(* IEC 61131-3 sources: BLM_BACKGROUND/src/PROGRAM_FILES/FB (part 5) *)

              //Modifica per gestione override come limitazione e non come percentuale
              ovr:=(i_sys_hwOvr_appo*i_sys_swOvr)/100;
              IF ovr>i_sys_tOVR THEN
                  ovr:=i_sys_tOVR;
              END_IF;
            //   {#ifdef PROFINET}
            //       {#ifndef ORBITALE}
                      IF TestVelHoldToRun()=TRUE AND i_sys_OPMODE=AUTOMODE AND FlgRiduzVelVGP=FALSE AND (TestMasterLavoro()=TRUE OR FlgPezzoInEsecuzione=TRUE) THEN
                          //Impostazione override per gestione hold TO run in automatico immediatamente al termine del primo start, così
                          //che al momento di iniziare la movimentazione degli assi l^override attivo sia già impostato al valore definito
                          //nel parametro Q4100
                          IF ovr>i_sys_override_HoldToRun_Auto THEN
                              ovr:=i_sys_override_HoldToRun_Auto;
                          END_IF;
                      END_IF;
            //       {#endif}  //Fine NO ORBITALE
            //   {#endif}	//Fine PROFINET
              IF i_sys_stopcond<>0 THEN
                //   {#ifdef PROFINET}
                      IF (i_Barriera=FALSE OR i_sys_BarrieraViolata=TRUE) AND TEMPO_ARRESTO_BARRIERA>0.01 THEN
                          //In caso di violazione della barriera di sicurezza se definita
                          //si attiva l^apposita rampa di decelerazione
                          Appo:=TEMPO_ARRESTO_BARRIERA;
                          AccelerazioneMaster:=1/Appo;
                      ELSE
                          AccelerazioneMaster:=i_sys_acc_master;
                      END_IF;
                //   {#else}  //Fine PROFINET
                      IF i_sys_BarrieraViolata=TRUE AND TEMPO_ARRESTO_BARRIERA>0.01 THEN
                          //In caso di violazione della barriera di sicurezza se definita
                          //si attiva l^apposita rampa di decelerazione
                          Appo:=TEMPO_ARRESTO_BARRIERA;
                          AccelerazioneMaster:=1/Appo;
                      ELSE
                          AccelerazioneMaster:=i_sys_acc_master;
                      END_IF;
                //   {#endif}  //Fine NO PROFINET
                  i_sys_ovr:=0;
                  CURRENT_STATE:=_FB_MCP483#STATE_MCP483_STOP_ASSI_MASTER;
              ELSE
                //   {#ifdef ORBITALE}
                //       {#ifdef DH4010}
                          i_sys_ovr:=ovr;
                    //   {#else}  //Fine DH4010
                          IF i_sys_OPMODE=AUTOMODE THEN
                              IF TestMasterLavoro()=TRUE THEN
                                  IF getBit(TO_DWORD(ReadTabStati(Riga:=rc, Colonna:=COL_RESERVED1, Programma:=I_SYS_Current_Prog, Tabella:=SINT#-1)), TO_USINT(BIT_NO_OVERRIDE))=TRUE THEN
                                      //Gestione forzatura OVERRIDE nel ciclo automatico nelle linee della tabella
                                      //stati dove e^ previsto (ad esempio per il taglio)
                                      i_sys_ovr_act:=100;
                                      i_sys_ovr:=100;
                                      masteraxis:=AsPositioningAxisRef(Axes[X1].masteraxis);
                                      masteraxis^._override.velocity:=100;
                                  ELSE
                                      i_sys_ovr:=ovr;
                                  END_IF;
                              ELSE
                                  //Primo start
                                //   {#ifdef FOUR_RUNNER_PLAUNO}
                                      IF i_sys_OverrideMarcatura=TRUE THEN
                                          //Forzatura override al 100% per mantenere costante la lunghezza della scritta
                                          i_sys_ovr_act:=100;
                                          i_sys_ovr:=100;
                                          masteraxis:=AsPositioningAxisRef(Axes[X1].masteraxis);
                                          masteraxis^._override.velocity:=100;
                                          //Axes[X1].masteraxis._override.velocity:=100;
                                      ELSE
                                          //Ripristiono override al termine della marcatura
                                          i_sys_ovr:=ovr;
                                      END_IF;
                                //   {#else}	//Fine FOUR_RUNNER_PLAUNO
                                      i_sys_ovr:=ovr;
                                //   {#endif};    //Fine NO FOUR_RUNNER_PLAUNO
                              END_IF;
                          ELSE
                              i_sys_ovr:=ovr;
                          END_IF;
                //       {#endif}  //Fine NO DH4010
                //   {#else}  //Fine ORBITALE
                      i_sys_ovr:=ovr;
                //   {#endif}  //Fine NO ORBITALE
                  CURRENT_STATE:=_FB_MCP483#STATE_MCP483_READ_OVR_2;
              END_IF;

            _FB_MCP483#STATE_MCP483_STOP_ASSI_MASTER:
              IF StopAssiMaster.outputState<>GENERAL_STATE#STATE_END THEN
                  StopAssiMaster(AccelerazioneMaster:=AccelerazioneMaster (* , ProssimoComando:=IMMEDIATELY*));
              ELSE
                  StopAssiMaster();
                  CURRENT_STATE:=_FB_MCP483#STATE_MCP483_READ_OVR_2;
              END_IF;

            _FB_MCP483#STATE_MCP483_READ_OVR_2:
               {::ifndef MCP_1900}
                  //Legge il II Override
                  i_sys_hwOVR2:=read_ovr2(mcpi_spindleoverride_a,mcpi_spindleoverride_b,mcpi_spindleoverride_c,mcpi_spindleoverride_d);
                  ovr2:=((i_sys_hwOvr2)/100) * ((i_sys_swOvr2)/100) * 100;
                  IF i_sys_stopcond<>0 THEN
                      i_sys_ovr2:=0;
                  ELSE
                      i_sys_ovr2:=ovr2;
                  END_IF;
               {::else}	//FINE NO MCP_1900
                  IF i_sys_stopcond<>0 THEN
                      i_sys_ovr2:=0;
                  ELSE
                      i_sys_ovr2:=100;
                  END_IF;
            {::endif} //FINE MCP_1900
              ovr2:=((i_sys_hwOvr2)/100) * ((i_sys_swOvr2)/100) * 100;
              IF i_sys_stopcond<>0 THEN
                  i_sys_ovr2:=0;
              ELSE
                  i_sys_ovr2:=ovr2;
              END_IF;
              //Assegnazione override all^asse master, per fare in modo di gestire la velocità
              //degli assi collegati in camma
              IF i_sys_stopcond=0 THEN
                  //Non deve essere attivo lo stop ciclo, in quanto in quella fase
                  //l^arresto dell master avviene con un normale comando di stop, associato
                  //alla rampa di decelerazione definita nella variabile AccelerazioneMaster
                  IF ABS(GetMasterOverride()-i_sys_ovr)>0.9 AND TestMasterVeloc()=TRUE THEN
                      //Al cambio di override corrisponde una immediata impostazione dell^accelerazione
                      //dell^asse master pari a 3 (quindi siamo a 0.3 secondi di rampa)
                      //Questo per evitare che ad ogni gradino venga causata sugli assi veri una
                      //accelerazione/decelerazione troppo elevata
                      IF ABS(GetMasterMaxAcceleration()-ACCELERATION_MASTER)>0.1 THEN
                          SetMasterMaxAcceleration(Value:=ACCELERATION_MASTER);
                      END_IF;
                  ELSE
                      //Senza nessun cambio di override si ripristina l^accelerazione standard del master
                      //molto elavata
                      IF ABS(GetMasterMaxAcceleration()-MAX_MASTER_ACCELERATION)>0.1 THEN
                          SetMasterMaxAcceleration(Value:=MAX_MASTER_ACCELERATION);
                      END_IF;
                  END_IF;
                  //Impostazione dell^override dell^asse master
                  IF ABS(GetMasterOverride()-i_sys_ovr_Act)>0.001 THEN
                      SetMasterVelocity(Value:=i_sys_ovr_Act);
                    //   {#ifdef RUNNER}
                    //       {#ifdef FOUR_RUNNER_PLAUNO}
                    //           {#ifndef PLAUNO_LIGHT}
                                masteraxis:=AsPositioningAxisRef(Axes[A1].masteraxis);
                                masteraxis^._override.velocity:=i_sys_ovr_Act;
                        //       {#endif} //FINE NO PLAUNO_LIGHT
                        //   {#endif}  //Fine FOUR_RUNNER_PLAUNO
                        //   {#ifdef B1_B2}
                              masteraxis:=AsPositioningAxisRef(Axes[B1].masteraxis);
                              masteraxis^._override.velocity:=i_sys_ovr_Act;
                    //       {#endif}  //Fine B1_B2
                    //   {#endif}  //Fine RUNNER
                  END_IF;
              ELSE
                  //Lo stop ciclo è attivo
                  IF TestMasterVeloc()=FALSE THEN
                      //Con stop ciclo attivo si imposta l^override desiderato quando il master si è fermato
                      IF ABS(GetMasterOverride()-i_sys_ovr_Act)>0.001 THEN
                          SetMasterVelocity(Value:=i_sys_ovr_Act);
                        //   {#ifdef RUNNER}
                        //       {#ifdef FOUR_RUNNER_PLAUNO}
                        //           {#ifndef PLAUNO_LIGHT}
                                      masteraxis:=AsPositioningAxisRef(Axes[A1].masteraxis);
                                      masteraxis^._override.velocity:=i_sys_ovr_Act;
                            //       {#endif} //FINE NO PLAUNO_LIGHT
                            //   {#endif}  //Fine FOUR_RUNNER_PLAUNO
                            //   {#ifdef B1_B2}
                                    masteraxis:=AsPositioningAxisRef(Axes[B1].masteraxis);
                                    masteraxis^._override.velocity:=i_sys_ovr_Act;
                        //       {#endif}  //Fine B1_B2
                        //   {#endif}  //Fine RUNNER
                      END_IF;
                  END_IF;
                  //Lo stop ciclo si esegue con l^accelerazione standard del master
                  IF ABS(GetMasterMaxAcceleration()-MAX_MASTER_ACCELERATION)>0.1 THEN
                      SetMasterMaxAcceleration(Value:=MAX_MASTER_ACCELERATION);
                  END_IF;
              END_IF;
              FOR i:=_FIRST_AXIS#FIRST_AXIS TO _FIRST_AXIS#FIRST_AXIS+_MAXIS#MAXAXIS-1 BY 1 DO
                  IF CheckIfTOactive(Axis:=i)=TRUE THEN
                      //Se l^asse non è in CAMMA
                      PosAx:=AsSynchronousAxisRef(Axes[i].PosAx);
                      Camma:= AsCamRef(PosAx^.StatusSynchronizedMotion.ActualCam);
                      IF   PosAx^.StatusSynchronizedMotion.FunctionState <>3 THEN
                          {::ifdef AL_BLM}
                              IF i=L1 THEN
                                  //Essendo L1 un asse del caricatore, non deve essere gestito normalmente
                                  //in quanto deve consentire il funzionamento del caricatore, anche quando
                                  //l^override è impostato a 0 in quanto il dispositivo è fuori posizione
                                  IF i_sys_stopcond=1 THEN
                                    ;
                                      PosAx^._override.velocity:=i_sys_ovr_act;
                                  ELSE
                                    ;
                                      PosAx^._override.velocity:=i_sys_hwovr;
                                  END_IF;
                              ELSE
                            //     //   {#ifdef ASSE_Z2}
                                      IF i=Z2 THEN
                                        PosAx:=AsSynchronousAxisRef(Axes[i].PosAx);
                                          IF i_sys_stopcond=1 THEN ;
                                            PosAx^._override.velocity:=i_sys_ovr_act;
                                          ELSE ;
                                            PosAx^._override.velocity:=100;
                                          END_IF;
                                      ELSE ;
                                            PosAx^._override.velocity:=i_sys_ovr_act;
                                      END_IF;
                                //   {#else}  //Fine ASSE_Z2
                                            PosAx^._override.velocity:=i_sys_ovr_act;
                                //   {#endif}  //Fine NO ASSE_Z2
                              END_IF;
                          {::else}  //Fine AL_BLM
                        //       {#ifdef EFLEX}
                                  IF i=W1 THEN
                                        PosAx:=AsSynchronousAxisRef(Axes[i].PosAx);
                                      IF (i_sys_OpMode=JOGMODE AND i_sys_activedevice=CMD_TAGLIO_EFLEX) OR
                                           (i_sys_OpMode=AUTOMODE AND PosizioneMaster()=POSIZIONE_MASTER_RFI) THEN
                                          //Asse W1 (trancia) non deve sentire override quando taglia con
                                          //il comando manuale
                                          PosAx^._override.velocity:=100;
                                      ELSE
                                          PosAx^._override.velocity:=i_sys_ovr_act;
                                      END_IF;
                                  ELSE
                                      //Gestione standard asse
                                      PosAx^._override.velocity:=i_sys_ovr_act;
                                  END_IF;
                            //   {#else}  //Fine EFLEX
                            //       {#ifdef RUNNER}
                            //           {#ifdef FOUR_RUNNER_PLAUNO}
                            //               {#ifdef B1_B2}
                                            //   IF {#ifndef PLAUNO_LIGHT}i=A1 OR i=A2 OR {#endif} i=B1 OR i=B2 THEN
                                            //       IF i_sys_ovr_act>0.1 THEN
                                            //           assi[i].PosAx._override.velocity:=100;
                                            //       ELSE
                                            //           assi[i].PosAx._override.velocity:=i_sys_ovr_act;
                                            //       END_IF;
                                            //   ELSE
                                            //       //Gestione standard asse
                                            //       assi[i].PosAx._override.velocity:=i_sys_ovr_act;
                                            //   END_IF;
                                        //   {#else}  //Fine B1_B2
                                        //       {#ifndef PLAUNO_LIGHT}
                                                  IF i=A1 OR i=A2 THEN
                                                    PosAx:=AsSynchronousAxisRef(Axes[i].PosAx);
                                                      IF i_sys_ovr_act>0.1 THEN ;
                                                          //PosAx^._override.velocity:=100;
                                                      ELSE ;
                                                          //PosAx^._override.velocity:=i_sys_ovr_act;
                                                      END_IF;
                                                  ELSE ;
                                            //   {#endif} //FINE NO PLAUNO_LIGHT
                                              //Gestione standard asse
                                                   // PosAx^._override.velocity:=i_sys_ovr_act;
                                            //   {#ifndef PLAUNO_LIGHT}
                                                  END_IF;
                                    //           {#endif}	//Fine PLAUNO_LIGHT
                                    //       {#endif}  //Fine NO B1_B2
                                    //   {#endif}  //Fine FOUR_RUNNER_PLAUNO
                                    //   {#ifdef THREE_RUNNER_TWO_RUNNER}
                                    //       {#ifdef B1_B2}
                                              IF i=A1 OR i=B1 OR i=B2 THEN
                                                PosAx:=AsSynchronousAxisRef(Axes[i].PosAx);
                                                  IF i_sys_ovr_act>0.1 THEN ;
                                                      //PosAx^._override.velocity:=100;
                                                  ELSE ;
                                                      //PosAx^._override.velocity:=i_sys_ovr_act;
                                                  END_IF;
                                              ELSE ;
                                                  //Gestione standard asse
                                                  //PosAx^._override.velocity:=i_sys_ovr_act;
                                              END_IF;
                                        //   {#else}  //Fine B1_B2
                                              IF i=A1 THEN
                                                  IF i_sys_ovr_act>0.1 THEN ;
                                                      //PosAx^._override.velocity:=100;
                                                  ELSE ;
                                                      //PosAx^._override.velocity:=i_sys_ovr_act;
                                                  END_IF;
                                              ELSE ;
                                                  //Gestione standard asse
                                                  //PosAx^._override.velocity:=i_sys_ovr_act;
                                              END_IF;
                                //           {#endif}  //Fine NO B1_B2
                                //       {#endif}  //Fine THREE_RUNNER_TWO_RUNNER
                                //   {#else}  //Fine RUNNER
                                      //Gestione standard asse
                                      //PosAx^._override.velocity:=i_sys_ovr_act;
                        //           {#endif}  //Fine NO RUNNER
                        //       {#endif}  //Fine NO EFLEX
                          {::endif}  //Fine NO AL_BLM
                          ;
                      END_IF;
                  END_IF;
              END_FOR;
              //Assegna l^override agli oggetti interpolatore
              {::ifndef ORBITALE}
                KinAxesX1_U2_def:= KinAxesX1_U2;
                X1_U2:= AsKinematicsRef(KinAxesX1_U2_def);
                X1_U2^._override.velocity:=i_sys_ovr_act;
              {::endif}  //Fine ORBITALE
                //{::ifndef ETURN}
                    // {::ifndef ORBITALE}
                    //   {::ifndef ELECTMRL}
                    //         KinAxesW3_W4_Q1_def:= KinAxesW3_W4_Q1;
                    //         W3_W4_Q1:= AsKinematicsRef(KinAxesW3_W4_Q1_def);
                    //       W3_W4_Q1^._override.velocity:=i_sys_ovr_act;
                    // //   {#else}
                    //         KinAxesW3_W4_W6_Q1_def:= KinAxesW3_W4_W6_Q1;
                    //         W3_W4_W6_Q1:= AsKinematicsRef(KinAxesW3_W4_W6_Q1_def);
                    //         W3_W4_W6_Q1^._override.velocity:=i_sys_ovr_act;
            //           {#endif} //FINE ELECTMRL
            //       {#endif}	//Fine ORBITALE
            //   {#endif}  //Fine ETURN
            //   {#ifdef INTERPOLA_Y1_X1}
                  //Y1_X1._override.velocity:=i_sys_ovr_act;//
            //   {#endif}    //Fine INTERPOLA_Y1_X1
            //   {#ifdef INTERPOLA_X1_Y1}
                  //X1_Y1._override.velocity:=i_sys_ovr_act;//
            //   {#endif}	//Fine INTERPOLA_X1_Y1
            //   {#ifdef INTERPOLA_X2_Y2}
                  //X2_Y2._override.velocity:=i_sys_ovr_act;//
            //   {#endif}	//Fine INTERPOLA_X2_Y2
            //   {#ifdef INTERPOLA_X3_X6}
                  //X3_X6._override.velocity:=i_sys_ovr_act;//
            //   {#endif}	//Fine INTERPOLA_X3_X6
            //   {#ifdef INTERPOLA_X2_X6}
                  //X2_X6._override.velocity:=i_sys_ovr_act;//
            //   {#endif}	//Fine INTERPOLA_X2_X6
            {::ifdef SLITTA_MOBILE_DX}
             KinAxesY1_U4_def:= KinAxesY1_U4;
             Y1_U4:= AsKinematicsRef(KinAxesY1_U4_def);
             Y1_U4^._override.velocity:=i_sys_ovr_act;
                  //Y1_U4._override.velocity:=i_sys_ovr_act;//
            {::endif}	//Fine SLITTA_MOBILE_DX
            //   {#ifdef SLITTA_MOBILE_SX}
                  //Y1_U5._override.velocity:=i_sys_ovr_act;//
            //   {#endif}	//Fine SLITTA_MOBILE_SX
            //    {::ifdef MATRICE_ELETTRICA}
            //       IF TestAxesY2()=TRUE THEN
            //           Y1_U4_Y2._override.velocity:=i_sys_ovr_act;//
            //            Y1_Y2._override.velocity:=i_sys_ovr_act;//
            //        END_IF;
            //    {::endif}  //Fine MATRICE_ELETTRICA
            //   {#ifdef SOLLEVAMENTO_SLITTA_SPALLAMENTO}
                //   Q1_V1_V4._override.velocity:=i_sys_ovr_act;//
                //   Q1_V1._override.velocity:=i_sys_ovr_act;
            //   {#endif}	//Fine SOLLEVAMENTO_SLITTA_SPALLAMENTO
               {::ifdef INTERPOLA_Q1_V1_Z1}
            KinAxesQ1_V1_Z1_def:= KinAxesQ1_V1_Z1;
            Q1_V1_Z1:= AsKinematicsRef(KinAxesY1_U4_def);
            Q1_V1_Z1^._override.velocity:=i_sys_ovr_act;
                  //Q1_V1_Z1._override.velocity:=i_sys_ovr_act;
               {::endif}    //Fine INTERPOLA_Q1_V1_Z1
              IF i_sys_current_prog>=0 THEN
                  //Rinfresca il MASTER
                  SetPosizioneMaster(Programma:=i_sys_current_prog);
              END_IF;
              CURRENT_AXIS:=_FIRST_AXIS#FIRST_AXIS-1;
              CURRENT_STATE:= _FB_MCP483#STATE_MCP483_LOOP_HOMING;

        _FB_MCP483#STATE_MCP483_LOOP_HOMING:
              FOR i:=CURRENT_AXIS+1 TO _MAXIS#MAXAXIS-1 BY 1 DO
                  IF TestToAttivo(Asse:=i)=TRUE THEN
                    PosAx:=AsSynchronousAxisRef(Axes[i].PosAx);
                      IF  Posax^.StatusWord.%x1 = TRUE THEN
                          IF Posax^.ErrorDetail.Reaction<>0 THEN
                              //Ferma tutti gli altri assi
                              i_sys_stopcond:=1;
                              IF Posax^.StatusWord.%X0=TRUE THEN
                                  Abort_All();
                              END_IF;
                          END_IF;
                      END_IF;

                      //Verifica eventuali errori di creazione della camma
                      IF PosAx^.StatusSynchronizedMotion.ActualMaster <> UDINT#0 THEN
                     // IF Axes[i].sincroasse.activemaster<> NULL THEN
                        Camma:= AsCamRef(Axes[i].Camma);
                            IF Camma^.StatusWord.%X1 =TRUE THEN
                            //IF Axes[i].Camma.error=YES THEN
                               IF Camma^.ErrorDetail.Reaction <> 0 THEN
                              //IF assi[i].Camma.errorreaction<>NONE THEN
                                  i_sys_stopcond:=1;
                                    IF Posax^.StatusWord.%X0=TRUE THEN
                                  //IF assi[i].Posax.control=ACTIVE THEN
                                      Abort_All();
                                  END_IF;
                              END_IF;
                          END_IF;
                      END_IF;
                      IF posax^.VirtualAxis.Mode = UDINT#0 THEN
                          IF pm[i].ma_verifica_num_serie_encoder=TRUE THEN
                              Axes[i].Homed:=Axes[i].numserieencoder=pm[i].ma_num_serie_encoder AND
                                                           Axes[i].numserieencoder>0 AND
                                                           PosAx^.StatusWord.%X5= TRUE AND
                                                           pm[i].ma_stato_index=2;
                          ELSE
                              Axes[i].Homed:=PosAx^.StatusWord.%X5=TRUE AND
                                                           pm[i].ma_stato_index=2;
                        ;  END_IF;
                      ELSE
                          IF PosAx^.StatusWord.%X5=TRUE THEN
                              //Asse virtuale l^asse viene indexato di default
                              pm[i].ma_stato_index:=SINT#0;
                              CURRENT_AXIS:=i;
                              CURRENT_STATE:=_FB_MCP483#STATE_MCP483_LOOP_HOMING_ABSOLUTE;
                              EXIT;
                          END_IF;
                      END_IF;
                  END_IF;
              END_FOR;
              IF CURRENT_STATE<>_FB_MCP483#STATE_MCP483_LOOP_HOMING_ABSOLUTE THEN
                  CURRENT_STATE:=_FB_MCP483#STATE_MCP483_CHECK_HOMING_ERRORS;
              END_IF;

            //   CURRENT_AXIS:=CURRENT_AXIS+1;
            //   IF CURRENT_AXIS<_MAXIS#MAXAXIS THEN
            //     PosAx:= AsSynchronousAxisRef(Axes[CURRENT_AXIS].Posax);
            //       IF TestToAttivo(Asse:=CURRENT_AXIS)=TRUE THEN
            //           IF Posax^.ErrorWord=TRUE THEN
            //             IF Posax^.ErrorDetail.Reaction<>0 THEN
            //               //IF assi[CURRENT_AXIS].Posax.errorreaction<>NONE THEN
            //                   //Ferma tutti gli altri assi
            //                   i_sys_stopcond:=1;
            //                   IF Posax^.StatusWord.%X0=TRUE THEN
            //                   //IF assi[CURRENT_AXIS].Posax.control=ACTIVE THEN
            //                       Abort_All();
            //                   END_IF;
            //               END_IF;
            //           END_IF;
            //           sincroasse:= AsSynchronousAxisRef( assi[CURRENT_AXIS].Sincroasse);
            //           IF Sincroasse^.ErrorWord=TRUE THEN
            //           //IF.error=YES THEN
            //             IF Sincroasse^.ErrorDetail.Reaction<>0 THEN
            //               //IF Sincroasse^.errorreaction<>NONE THEN
            //                   i_sys_stopcond:=1;
            //                   PosAx:= AsSynchronousAxisRef(Axes[i].Posax);
            //                   IF Posax^.StatusWord.%X0=TRUE THEN
            //                       Abort_All();
            //                   END_IF;
            //               END_IF;
            //           END_IF;
            //           //Verifica eventuali errori di creazione della camma
            //           sincroasse:= AsSynchronousAxisRef(Axes[CURRENT_AXIS].sincroasse);
            //           IF sincroasse^.StatusSynchronizedMotion.ActualMaster <> UDINT#0 THEN
            //           //IF Axes[CURRENT_AXIS].sincroasse.activemaster<>NULL THEN
            //           Camma:= AsCamRef(Axes[i].Camma);
            //           IF Camma^.ErrorWord=TRUE THEN
            //           //IF Axes[i].Camma.error=YES THEN
            //              IF Camma^.ErrorDetail.Reaction <> 0 THEN
            //               //IF assi[CURRENT_AXIS].Camma.error=YES THEN
            //                   //IF assi[CURRENT_AXIS].Camma.errorreaction<>NONE THEN
            //                       i_sys_stopcond:=1;
            //                       IF assi[CURRENT_AXIS].Posax.control=ACTIVE THEN
            //                           Abort_All();
            //                       END_IF;
            //                   END_IF;
            //               END_IF;
            //           END_IF;
            //           IF Axes[CURRENT_AXIS].posax.typeofaxis<>VIRTUAL_AXIS THEN
            //               IF pm[CURRENT_AXIS].ma_verifica_num_serie_encoder=TRUE THEN
            //                   Axes[CURRENT_AXIS].Homed:=Axes[CURRENT_AXIS].numserieencoder=pm[CURRENT_AXIS].ma_num_serie_encoder AND
            //                                                Axes[CURRENT_AXIS].numserieencoder>0 AND
            //                                                Axes[CURRENT_AXIS].PosAx.positioningstate.homed=YES AND
            //                                                pm[CURRENT_AXIS].ma_stato_index=2;
            //               ELSE
            //                   Axes[CURRENT_AXIS].Homed:=Axes[CURRENT_AXIS].PosAx.positioningstate.homed=YES AND
            //                                                pm[CURRENT_AXIS].ma_stato_index=2;
            //               END_IF;
            //           ELSE
            //               IF Axes[CURRENT_AXIS].PosAx.positioningstate.homed<>YES THEN
            //                   //Asse virtuale l^asse viene indexato di default
            //                   pm[CURRENT_AXIS].ma_stato_index:=0;
            //                   CURRENT_STATE:=STATE_MCP483_LOOP_HOMING_HOMING_ABSOLUTE;
            //               END_IF;
            //           END_IF;
            //       END_IF;
            //   ELSE
            //       CURRENT_STATE:=_FB_MCP483#STATE_MCP483_CHECK_HOMING_ERRORS;
            //   END_IF;

          _FB_MCP483#STATE_MCP483_LOOP_HOMING_ABSOLUTE:
              IF Homing_Absolute.outputState<>GENERAL_STATE#STATE_END THEN
                  Homing_absolute(Asse:=CURRENT_AXIS, Position:=0);
              ELSE
                  Homing_absolute();
                  Axes[CURRENT_AXIS].homed:=TRUE;
                  CURRENT_STATE:=_FB_MCP483#STATE_MCP483_LOOP_HOMING;
              END_IF;

          _FB_MCP483#STATE_MCP483_CHECK_HOMING_ERRORS:
            //   {#ifdef INTERPOLA_Y1_X1}
                //   IF Y1_X1.error=YES THEN %%%%
                //       IF Y1_X1.errorreaction<>NONE THEN
                //           //Ferma tutti gli altri assi
                //           i_sys_stopcond:=1;
                //           IF Y1_X1.linearPathCommand.state=ACTIVE THEN //OT.StatusWord.%X8
                //               iret:=Push_error(code:=ERR_VETT_Y1_X1, Arresto:=TRUE);
                //           ELSE
                //               iret:=Push_error(code:=ERR_VETT_Y1_X1, Arresto:=FALSE);
                //           END_IF;
                //       END_IF;
                //   END_IF;
            //   {#endif}	//Fine INTERPOLA_Y1_X1
            //   {#ifdef INTERPOLA_X1_Y1}
                //   IF X1_Y1.error=YES AND X1_Y1.errorreaction<>NONE AND I_Barriera=TRUE AND i_sys_BarrieraViolata=FALSE THEN %%%%
                //       //Ferma tutti gli altri assi
                //       i_sys_stopcond:=1;
                //       IF X1_Y1.linearPathCommand.state=ACTIVE THEN
                //           iret:=Push_error(code:=ERR_VETT_X1_Y1, Arresto:=TRUE);
                //       ELSE
                //           iret:=Push_error(code:=ERR_VETT_X1_Y1, Arresto:=FALSE);
                //       END_IF;
                //   END_IF;
            //   {#endif}	//Fine INTERPOLA_X1_Y1
            //   {#ifdef INTERPOLA_X2_Y2}
                //   IF X2_Y2.error=YES AND X2_Y2.errorreaction<>NONE AND I_Barriera=TRUE AND i_sys_BarrieraViolata=FALSE THEN %%%%

                //       //Ferma tutti gli altri assi
                //       i_sys_stopcond:=1;
                //       IF X2_Y2.linearPathCommand.state=ACTIVE THEN
                //           iret:=Push_error(code:=ERR_VETT_X2_Y2, Arresto:=TRUE);
                //       ELSE
                //           iret:=Push_error(code:=ERR_VETT_X2_Y2, Arresto:=FALSE);
                //       END_IF;
                //   END_IF;
            //   {#endif}	//Fine INTERPOLA_X1_Y1
            //   {#ifdef INTERPOLA_X3_X6}
                //   IF X3_X6.error=YES AND X3_X6.errorreaction<>NONE AND I_Barriera=TRUE AND i_sys_BarrieraViolata=FALSE THEN %%%%
                //       //Ferma tutti gli altri assi
                //       i_sys_stopcond:=1;
                //       IF X3_X6.linearPathCommand.state=ACTIVE THEN
                //           iret:=Push_error(code:=ERR_VETT_X3_X6, Arresto:=TRUE);
                //       ELSE
                //           iret:=Push_error(code:=ERR_VETT_X3_X6, Arresto:=FALSE);
                //       END_IF;
                //   END_IF;
            //   {#endif}	//Fine INTERPOLA_X3_X6
            //   {#ifdef INTERPOLA_X2_X6}
                //   IF X2_X6.error=YES AND X2_X6.errorreaction<>NONE AND I_Barriera=TRUE AND i_sys_BarrieraViolata=FALSE THEN %%%%
                //       //Ferma tutti gli altri assi
                //       i_sys_stopcond:=1;
                //       IF X2_X6.linearPathCommand.state=ACTIVE THEN
                //           iret:=Push_error(code:=ERR_VETT_X2_X6, Arresto:=TRUE);
                //       ELSE
                //           iret:=Push_error(code:=ERR_VETT_X2_X6, Arresto:=FALSE);
                //       END_IF;
                //   END_IF;
            //   {#endif}	//Fine INTERPOLA_X2_X6
            //   {#ifdef SLITTA_MOBILE_DX}

            //   {#endif}	//Fine SLITTA_MOBILE_DX
            //   {#ifdef SLITTA_MOBILE_SX}
                //   IF Y1_U5.error=YES THEN
                //       IF Y1_U5.errorreaction<>NONE THEN
                //           //Ferma tutti gli altri assi
                //           i_sys_stopcond:=1;
                //           IF Y1_U5.linearPathCommand.state=ACTIVE THEN
                //               iret:=Push_error(code:=ERR_VETT_Y1_U4, Arresto:=TRUE);
                //           ELSE
                //               iret:=Push_error(code:=ERR_VETT_Y1_U4, Arresto:=FALSE);
                //           END_IF;
                //       END_IF;
                //   END_IF;
            //   {#endif}  //Fine SLITTA_MOBILE_SX
            //   {#ifndef ORBITALE}
                //   IF X1_U2.error=YES THEN
                //       IF X1_U2.errorreaction<>NONE THEN
                //           //Ferma tutti gli altri assi
                //           i_sys_stopcond:=1;
                //           IF X1_U2.linearPathCommand.state=ACTIVE THEN
                //               iret:=Push_error(code:=ERR_VECT_CARRO_ANIMA, Arresto:=TRUE);
                //           ELSE
                //               iret:=Push_error(code:=ERR_VECT_CARRO_ANIMA, Arresto:=FALSE);
                //           END_IF;
                //       END_IF;
                //   END_IF;
            //   {#endif}  //Fine NO ORBITALE
            //   {#ifndef ETURN}
            //       {#ifndef ORBITALE}
            //           {#ifndef ELECTMRL}
                        //   IF W3_W4_Q1.error=YES THEN
                        //       IF W3_W4_Q1.errorreaction<>NONE THEN
                        //           //Ferma tutti gli altri assi
                        //           i_sys_stopcond:=1;
                        //           IF W3_W4_Q1.linearPathCommand.state=ACTIVE THEN
                        //               iret:=Push_error(code:=ERR_VECT_MORSA_RULLI_Q, Arresto:=TRUE);
                        //           ELSE
                        //               iret:=Push_error(code:=ERR_VECT_MORSA_RULLI_Q, Arresto:=FALSE);
                        //           END_IF;
                        //       END_IF;
                        //   END_IF;
                    //   {#else}    //FINE NO ELECTMRL
                        //   IF W3_W4_W6_Q1.error=YES THEN
                        //       IF W3_W4_W6_Q1.errorreaction<>NONE THEN
                        //           //Ferma tutti gli altri assi
                        //           i_sys_stopcond:=1;
                        //           IF W3_W4_W6_Q1.linearPathCommand.state=ACTIVE THEN
                        //               iret:=Push_error(code:=ERR_VECT_MORSA_RULLI_Q, Arresto:=TRUE);
                        //           ELSE
                        //               iret:=Push_error(code:=ERR_VECT_MORSA_RULLI_Q, Arresto:=FALSE);
                        //           END_IF;
                        //       END_IF;
                        //   END_IF;
            //           {#endif} //FINE ELECTMRL
            //       {#endif}  //Fine NO ORBITALE
            //   {#endif}  //Fine NO ETURN
            //   {#ifdef MATRICE_ELETTRICA}
                //   IF TestAxesY2()=TRUE THEN
                //       IF Y1_U4_Y2.error=YES THEN
                //           IF Y1_U4_Y2.errorreaction<>NONE THEN
                //               //Ferma tutti gli altri assi
                //               i_sys_stopcond:=1;
                //               IF Y1_U4_Y2.linearPathCommand.state=ACTIVE THEN
                //                   iret:=Push_error(code:=ERR_VECT_Y1_U4_Y2, Arresto:=TRUE);
                //               ELSE
                //                   iret:=Push_error(code:=ERR_VECT_Y1_U4_Y2, Arresto:=FALSE);
                //               END_IF;
                //           END_IF;
                //       END_IF;
                //       IF Y1_Y2.error=YES THEN
                //           IF Y1_Y2.errorreaction<>NONE THEN
                //               //Ferma tutti gli altri assi
                //               i_sys_stopcond:=1;
                //               IF Y1_Y2.linearPathCommand.state=ACTIVE THEN
                //                   iret:=Push_error(code:=ERR_VECT_Y1_Y2, Arresto:=TRUE);
                //               ELSE
                //                   iret:=Push_error(code:=ERR_VECT_Y1_Y2, Arresto:=FALSE);
                //               END_IF;
                //           END_IF;
                //       END_IF;
                //   END_IF;
            //   {#endif}  //Fine MATRICE_ELETTRICA
            //   {#ifdef SOLLEVAMENTO_SLITTA_SPALLAMENTO}
                //   IF Q1_V1_V4.error=YES THEN
                //       IF Q1_V1_V4.errorreaction<>NONE THEN
                //           //Ferma tutti gli altri assi
                //           i_sys_stopcond:=1;
                //           IF Q1_V1_V4.linearPathCommand.state=ACTIVE THEN
                //               iret:=Push_error(code:=ERR_VECT_Q_V1_V4, Arresto:=TRUE);
                //           ELSE
                //               iret:=Push_error(code:=ERR_VECT_Q_V1_V4, Arresto:=FALSE);
                //           END_IF;
                //       END_IF;
                //   END_IF;
                //   IF Q1_V1.error=YES THEN
                //       IF Q1_V1.errorreaction<>NONE THEN
                //           //Ferma tutti gli altri assi
                //           i_sys_stopcond:=1;
                //           IF Q1_V1.linearPathCommand.state=ACTIVE THEN
                //               iret:=Push_error(code:=ERR_VECT_Q_V1_V4, Arresto:=TRUE);
                //           ELSE
                //               iret:=Push_error(code:=ERR_VECT_Q_V1_V4, Arresto:=FALSE);
                //           END_IF;
                //       END_IF;
                //   END_IF;
            //   {#endif}	//Fine SOLLEVAMENTO_SLITTA_SPALLAMENTO

            //    {::ifdef INTERPOLA_Q1_V1_Z1}
                        Q1_V1_Z1:= AsKinematicsRef(KinAxesQ1_V1_Z1_def);
                       IF Q1_V1_Z1^.StatusWord.%X1=TRUE THEN
                          IF Q1_V1_Z1^.ErrorDetail.Reaction<>0 THEN
                          //Ferma tutti gli altri assi
                          i_sys_stopcond:=1;
                          IF Q1_V1_Z1^.StatusWord.%X8 THEN
                              iret:=Push_error(code:=ERR_VECT_TESTA_Q_T, Arresto:=TRUE);
                          ELSE
                              iret:=Push_error(code:=ERR_VECT_TESTA_Q_T, Arresto:=FALSE);
                          END_IF;
                      END_IF;
                  END_IF;
            //    {::endif}	//Fine INTERPOLA_Q1_V1_Z1
              IF i_sys_OPMODE=JOGMODE AND
                   i_sys_activedevice<FIRST_COMPLEX_OPERATION AND
                   TaskCicliAttivo THEN
                  (*dwret:=_resetTaskId(_task.motiontask_CICLI);*)
                  CURRENT_STATE:=_FB_MCP483#STATE_MCP483_ELIMINATE_HOMING_COMMANDS;
              ELSE
                  CURRENT_STATE:=_FB_MCP483#STATE_MCP483_GEST_JOG;
              END_IF;

          _FB_MCP483#STATE_MCP483_ELIMINATE_HOMING_COMMANDS:
              IF EliminaCodaComandi.outputState<>GENERAL_STATE#STATE_END THEN
                  EliminaCodaComandi();
              ELSE
                  EliminaCodaComandi();
                  i_sys_stopcond:=0;
                  TaskCicliAttivo:=FALSE;
                  CURRENT_STATE:=_FB_MCP483#STATE_MCP483_GEST_JOG;
              END_IF;

        _FB_MCP483#STATE_MCP483_GEST_JOG:
              //Gestisce il movimento in JOG
              IF i_sys_OPMODE=JOGMODE AND i_sys_activedevice>=_FIRST_AXIS#FIRST_AXIS AND i_sys_STOPCOND=0 THEN
                  //Verifica che non sia rimasto nessun asse in movimento
                  IF i_sys_activedevice>=_FIRST_AXIS#FIRST_AXIS AND i_sys_Activedevice<_MAXIS#MAXAXIS+_FIRST_AXIS#FIRST_AXIS THEN
                      //Verifica che non sia rimasto nessun asse in movimento
                      IF i_sys_activedevice>=_FIRST_AXIS#FIRST_AXIS AND i_sys_Activedevice<_MAXIS#MAXAXIS+_FIRST_AXIS#FIRST_AXIS THEN
                          //E^ un asse
                          // verifica e gestisce il JOG per assi reali
                        //   {#ifdef BLOCCAGGIO_DX}
                              IF i_sys_activedevice=W3 THEN
                                  AppoDirezione:=SN;
                              ELSE
                                  AppoDirezione:=SN_SP;
                              END_IF;
                        //   {#else}  //Fine BLOCCAGGIO_DX
                              AppoDirezione:=SN_SP;
                        //   {#endif}  //Fine NO BLOCCAGGIO_DX
                          CURRENT_STATE:=_FB_MCP483#STATE_MCP483_GEST_JOG_SET_CONDITION_MOVE_AXIS;
                      ELSE
                          IF i_sys_activedevice>=FIRST_DEVICE AND i_sys_Activedevice<FIRST_DEVICE+_MAXDEVICES#MAXDEVICES THEN
                              //E^ un dispositivo
                              CURRENT_AXIS:=_FIRST_AXIS#FIRST_AXIS-1;
                              CURRENT_STATE:=_FB_MCP483#STATE_MCP483_GEST_JOG_LOOP_AXIS_RESET_MOTION;
                          ELSE
                              IF TaskCicliAttivo=FALSE THEN
                                  //Comandi manuali complessi
                                  CURRENT_STATE:=_FB_MCP483#STATE_MCP483_GEST_JOG_TASK_ACTIVE;
                              ELSE
                                  CURRENT_AXIS:=_FIRST_AXIS#FIRST_AXIS-1;
                                  CURRENT_STATE:=_FB_MCP483#STATE_MCP483_GEST_JOG_LOOP_STEPS_ELIMINATE_COMMANDS;
                              END_IF;
                          END_IF;
                      END_IF;
                  ELSE
                      CURRENT_AXIS:=_FIRST_AXIS#FIRST_AXIS-1;
                      CURRENT_STATE:=_FB_MCP483#STATE_MCP483_GEST_JOG_LOOP_STEPS_ELIMINATE_COMMANDS;
                  END_IF;
              ELSE
                  CURRENT_AXIS:=_FIRST_AXIS#FIRST_AXIS-1;
                  CURRENT_STATE:=_FB_MCP483#STATE_MCP483_GEST_JOG_LOOP_STEPS_ELIMINATE_COMMANDS;
              END_IF;

          _FB_MCP483#STATE_MCP483_GEST_JOG_SET_CONDITION_MOVE_AXIS:
              IF Set_Condizione_Move_Asse.outputState<>GENERAL_STATE#STATE_END THEN
                  SET_Condizione_Move_Asse(Asse:=i_sys_activedevice);
              ELSE
                  SET_Condizione_Move_Asse();
                  IF OK_Condizione_Move_Asse(Asse:=i_sys_activedevice, Direzione:=AppoDirezione)=TRUE THEN
                      reset_trace(Code:=TRC_SAFETY_JOG_DEVICES);
                      IF i_sys_activedevice>=_FIRST_AXIS#FIRST_AXIS AND i_sys_Activedevice<_MAXIS#MAXAXIS+_FIRST_AXIS#FIRST_AXIS THEN
                          IF TestAssePronto(Asse:=i_sys_activedevice)=FALSE THEN
                              CURRENT_STATE:=_FB_MCP483#STATE_MCP483_GEST_JOG_ENABLE_AXIS_BLM;
                          ELSE
                              StatePower:=TRUE;
                              CURRENT_STATE:=_FB_MCP483#STATE_MCP483_GEST_JOG_CHECK_ENABLE_AXIS_BLM;
                          END_IF;
                      ELSE
                          CURRENT_STATE:=_FB_MCP483#STATE_MCP483_GEST_JOG_CHECK_ENABLE_AXIS_BLM;
                      END_IF;
                  ELSE
                      TaskCicliAttivo:=FALSE;
                      CURRENT_AXIS:=_FIRST_AXIS#FIRST_AXIS-1;
                      CURRENT_STATE:=_FB_MCP483#STATE_MCP483_GEST_JOG_LOOP_STEPS_ELIMINATE_COMMANDS;
                  END_IF;
              END_IF;

          _FB_MCP483#STATE_MCP483_GEST_JOG_ENABLE_AXIS_BLM:
              IF EnableAxisBLM.outputState<>GENERAL_STATE#STATE_END THEN
                  EnableAxisBlm(Axis:=Axes[i_sys_activedevice].PosAx,
                                              NumeroAsse:=i_sys_activedevice
                                              (*ModoAttesa:=IMMEDIATELY*));
              ELSE
                  EnableAxisBlm();
                  StatePower:=FALSE;
                  CURRENT_STATE:=_FB_MCP483#STATE_MCP483_GEST_JOG_CHECK_ENABLE_AXIS_BLM;
              END_IF;

          _FB_MCP483#STATE_MCP483_GEST_JOG_CHECK_ENABLE_AXIS_BLM:
              IF StatePower=TRUE THEN ;
                // //   {#ifdef PINZA_ELETTRICA}%%%%
                //     PosAx:=AsSynchronousAxisRef(Axes[W1].PosAx);
                //       IF i_sys_activedevice=W1 THEN
                //           IF PosAx^.StatusWord.%X7 THEN
                //               //Impostazione coppia pinza chiusa
                //               CURRENT_STATE:=_FB_MCP483#STATE_MCP483_GEST_JOG_ENABLE_COUPLE_W1_GENERIC;
                //           ELSE
                //             //   {#ifdef ELECTXL}
                //                   //Movimento manuale pinza a coppia ridotta (di calibrazione)
                //                   CURRENT_STATE:=_FB_MCP483#STATE_MCP483_GEST_JOG_ENABLE_PAIR_W1_ELECTXL;
                //             //   {#else}
                //             //       {#ifdef ETURN_MR}
                //                       //Movimento manuale pinza a coppia massima
                //                       CURRENT_STATE:=_FB_MCP483#STATE_MCP483_GEST_JOG_DISABLE_COUPLE_W1_ETURN;
                //                 //   {#else}
                //                       CURRENT_STATE:=_FB_MCP483#STATE_MCP483_GEST_JOG_JOG_ASSE;
                //             //       {#endif};
                //             //   {#endif};
                //           END_IF;
                //       ELSE
                //           CURRENT_STATE:=_FB_MCP483#STATE_MCP483_GEST_JOG_JOG_ASSE;
                //       END_IF;
                // //   {#else}
                //       CURRENT_STATE:=_FB_MCP483#STATE_MCP483_GEST_JOG_JOG_ASSE;
                // //   {#endif};
              ELSE
                  TaskCicliAttivo:=FALSE;
                  CURRENT_AXIS:=_FIRST_AXIS#FIRST_AXIS-1;
                  CURRENT_STATE:=_FB_MCP483#STATE_MCP483_GEST_JOG_LOOP_STEPS_ELIMINATE_COMMANDS;
              END_IF;

          _FB_MCP483#STATE_MCP483_GEST_JOG_ENABLE_COUPLE_W1_GENERIC:
          ;  //   {#ifdef PINZA_ELETTRICA}
                //   IF EnableAsseInCoppia.outputState<>GENERAL_STATE#STATE_END THEN %%%%
                //       EnableAsseInCoppia(Coppia:=i_sys_CoppiaPinzaChiusa, NumeroAsse:=W1, Attesa:=FALSE);
                //   ELSE
                //       EnableAsseInCoppia();
                //       CURRENT_STATE:=_FB_MCP483#STATE_MCP483_GEST_JOG_JOG_ASSE;
                //   END_IF;
            //   {#endif};

          _FB_MCP483#STATE_MCP483_GEST_JOG_ENABLE_PAIR_W1_ELECTXL:
            ;//   {#ifdef ELECTXL}
                //   IF EnableAsseInCoppia.outputState<>GENERAL_STATE#STATE_END THEN %%%%
                //       EnableAsseInCoppia(Coppia:=BlmMxToolsOffPezzo[W1].CoppiaRidotta*10,
                //                                            NumeroAsse:=W1,
                //                                            Attesa:=FALSE);
                //   ELSE
                //       EnableAsseInCoppia();
                //       CURRENT_STATE:=_FB_MCP483#STATE_MCP483_GEST_JOG_JOG_ASSE;
                //   END_IF;
            //   {#endif};

          _FB_MCP483#STATE_MCP483_GEST_JOG_DISABLE_COUPLE_W1_ETURN:
            //   {#ifdef ETURN_MR}
                  IF DisableAsseInCoppia.outputState<>GENERAL_STATE#STATE_END THEN
                      DisableAsseInCoppia(NumeroAsse:=W1, Verifica:=FALSE);
                  ELSE
                      DisableAsseInCoppia();
                      CURRENT_STATE:=_FB_MCP483#STATE_MCP483_GEST_JOG_JOG_ASSE;
                  END_IF;
            //   {#endif};

          _FB_MCP483#STATE_MCP483_GEST_JOG_JOG_ASSE:
              IF Jog_Asse.outputState<>GENERAL_STATE#STATE_END THEN
                  Jog_Asse(Asse:=i_sys_activedevice);
              ELSE
                  Jog_Asse();
                  TaskCicliAttivo:=FALSE;
                  CURRENT_AXIS:=_FIRST_AXIS#FIRST_AXIS-1;
                  CURRENT_STATE:=_FB_MCP483#STATE_MCP483_GEST_JOG_LOOP_STEPS_ELIMINATE_COMMANDS;
              END_IF;

          _FB_MCP483#STATE_MCP483_GEST_JOG_LOOP_AXIS_RESET_MOTION:
              CURRENT_AXIS:=CURRENT_AXIS+1;
              IF CURRENT_AXIS<_MAXIS#MAXAXIS THEN
                  IF TestDispConAsse(Disp:=i_sys_activedevice, Asse:=CURRENT_AXIS)=FALSE THEN
                      //Verifica che la movimentazione del dispositivo non debba anche essere associata ad una posizionamento di un asse,
                      //in tale caso non sarà possibile effettuare il reset di sicurezza in quanto si annullerebbe il necessario
                      //posizionamento dell^asse
                      PosAx:= AsSynchronousAxisRef(Axes[CURRENT_AXIS].PosAx);
                      PosAx:=AsSynchronousAxisRef(Axes[CURRENT_AXIS].posax);
                      IF PosAx^.StatusPositioning.Distance >0.01 AND posax^.simulation.Mode=UDINT#0 THEN
                          CURRENT_STATE:=_FB_MCP483#STATE_MCP483_GEST_JOG_RESET_MOTION_RESET_AXIS;
                      END_IF;
                  END_IF;
              ELSE
                  CURRENT_STATE:=_FB_MCP483#STATE_MCP483_GEST_JOG_SET_CONDITION_MOVE_DEVICE ;
              END_IF;

          _FB_MCP483#STATE_MCP483_GEST_JOG_RESET_MOTION_RESET_AXIS:
              IF ResetMotionResetAxis.outputState<>GENERAL_STATE#STATE_END THEN
                  //Per sicurezza si resettano gli assi che hanno ancora un percorso residuo
                  ResetMotionResetAxis(Asse:=CURRENT_AXIS, Attesa:=FALSE);
              ELSE
                  ResetMotionResetAxis();
                  CURRENT_STATE:=_FB_MCP483#STATE_MCP483_GEST_JOG_LOOP_AXIS_RESET_MOTION;
              END_IF;

          _FB_MCP483#STATE_MCP483_GEST_JOG_SET_CONDITION_MOVE_DEVICE :
              IF Set_Condizione_Move_Dispositivo.outputState<>GENERAL_STATE#STATE_END THEN
                  SET_Condizione_Move_Dispositivo(i_sys_activedevice);
              ELSE
                  SET_Condizione_Move_Dispositivo();
                  IF R_Plus.Q=TRUE AND Clk_minus=FALSE THEN
                      IF i_sys_monitoring<>0 OR i_sys_Accesslevel<=ACCESS_MANUTENTORE OR SbloccaMonitoring(Asse:=i_sys_Activedevice) THEN
                          Esito:=OK_Condizione_Move_Dispositivo(Dispositivo:=i_sys_activedevice,
                                                                                                      Stato:=LAVORO,
                                                                                                      TastoPiu:=TRUE,
                                                                                                      TastoMeno:=FALSE);
                          IF Esito=TRUE THEN
                              reset_trace(Code:=TRC_SAFETY_JOG_DEVICES);
                              CURRENT_STATE:=_FB_MCP483#STATE_MCP483_GEST_JOG_MOVE_DEVICE ;
                          ELSE
                              TaskCicliAttivo:=FALSE;
                              CURRENT_AXIS:=_FIRST_AXIS#FIRST_AXIS-1;
                              CURRENT_STATE:=_FB_MCP483#STATE_MCP483_GEST_JOG_LOOP_STEPS_ELIMINATE_COMMANDS;
                          END_IF;
                      ELSE
                          TaskCicliAttivo:=FALSE;
                          set_trace(Code:=TRC_JOG_NON_IN_MONITORING);
                          CURRENT_AXIS:=_FIRST_AXIS#FIRST_AXIS-1;
                          CURRENT_STATE:=_FB_MCP483#STATE_MCP483_GEST_JOG_LOOP_STEPS_ELIMINATE_COMMANDS;
                      END_IF;
                  ELSE
                      IF R_Minus.Q=TRUE AND Clk_plus=FALSE THEN
                          IF i_sys_monitoring<>0 OR i_sys_Accesslevel<=ACCESS_MANUTENTORE OR SbloccaMonitoring(Asse:=i_sys_Activedevice) THEN
                              Esito:=OK_Condizione_Move_Dispositivo(Dispositivo:=i_sys_activedevice,
                                                                                                          Stato:=RIPOSO,
                                                                                                          TastoPiu:=FALSE,
                                                                                                          TastoMeno:=TRUE);
                              IF Esito=TRUE THEN
                                  reset_trace(Code:=TRC_SAFETY_JOG_DEVICES);
                                  CURRENT_STATE:=_FB_MCP483#STATE_MCP483_GEST_JOG_MOVE_DEVICE_REST;
                              ELSE
                                  TaskCicliAttivo:=FALSE;
                                  CURRENT_AXIS:=_FIRST_AXIS#FIRST_AXIS-1;
                                  CURRENT_STATE:=_FB_MCP483#STATE_MCP483_GEST_JOG_LOOP_STEPS_ELIMINATE_COMMANDS;
                              END_IF;
                          ELSE
                              TaskCicliAttivo:=FALSE;
                              set_trace(Code:=TRC_JOG_NON_IN_MONITORING);
                              CURRENT_AXIS:=_FIRST_AXIS#FIRST_AXIS-1;
                              CURRENT_STATE:=_FB_MCP483#STATE_MCP483_GEST_JOG_LOOP_STEPS_ELIMINATE_COMMANDS;
                          END_IF;
                      ELSE
                          IF Clk_minus=FALSE AND Clk_plus=FALSE THEN
                              IF Disp[i_sys_activedevice].PresenzaCostante=TRUE THEN
                                  WriteDigitalOutput(NumOutput:=Disp[i_sys_activedevice].out_lavoro, Value:=FALSE);
                                  WriteDigitalOutput(NumOutput:=Disp[i_sys_activedevice].out_riposo, Value:=FALSE);
                              END_IF;
                              reset_trace(Code:=TRC_JOG_NON_IN_MONITORING);
                              TaskCicliAttivo:=FALSE;
                              CURRENT_AXIS:=_FIRST_AXIS#FIRST_AXIS-1;
                              CURRENT_STATE:=_FB_MCP483#STATE_MCP483_GEST_JOG_LOOP_STEPS_ELIMINATE_COMMANDS;
                          ELSE
                              IF Disp[i_sys_activedevice].spegnimentouscita=TRUE THEN
                                  IF Disp[i_sys_activedevice].Stato=Disp[i_sys_activedevice].StatoRichiesto THEN
                                      WriteDigitalOutput(NumOutput:=Disp[i_sys_activedevice].out_lavoro, Value:=FALSE);
                                      WriteDigitalOutput(NumOutput:=Disp[i_sys_activedevice].out_riposo, Value:=FALSE);
                                  END_IF;
                              END_IF;
                              TaskCicliAttivo:=FALSE;
                              CURRENT_AXIS:=_FIRST_AXIS#FIRST_AXIS-1;
                              CURRENT_STATE:=_FB_MCP483#STATE_MCP483_GEST_JOG_LOOP_STEPS_ELIMINATE_COMMANDS;
                          END_IF;
                      END_IF;
                  END_IF;
              END_IF;

          _FB_MCP483#STATE_MCP483_GEST_JOG_MOVE_DEVICE :
              IF MuoviDispositivo.outputState<>GENERAL_STATE#STATE_END THEN
                  MuoviDispositivo(Dispositivo:=i_sys_activedevice, Stato:=LAVORO);
              ELSE
                  MuoviDispositivo();
                  CURRENT_STATE:=_FB_MCP483#STATE_MCP483_GEST_JOG_LOOP_STEPS_ELIMINATE_COMMANDS;
              END_IF;

          _FB_MCP483#STATE_MCP483_GEST_JOG_MOVE_DEVICE_REST:
              IF MuoviDispositivo.outputState<>GENERAL_STATE#STATE_END THEN
                  MuoviDispositivo(Dispositivo:=i_sys_activedevice, Stato:=RIPOSO);
              ELSE
                  MuoviDispositivo();
                  CURRENT_AXIS:=_FIRST_AXIS#FIRST_AXIS-1;
                  CURRENT_STATE:=_FB_MCP483#STATE_MCP483_GEST_JOG_LOOP_STEPS_ELIMINATE_COMMANDS;
              END_IF;

          _FB_MCP483#STATE_MCP483_GEST_JOG_TASK_ACTIVE:
              IF TaskCicliAttivo=FALSE THEN
                  //Comandi manuali complessi
                  IF i_sys_activedevice>=FIRST_COMPLEX_OPERATION AND
                       i_sys_activedevice<>C_DISATTIVAZIONE_BOOSTER_X1 AND
                       i_sys_activedevice<>C_IMPOSTAZIONI_ASSI_DISATTIVABILI AND
                       i_sys_activedevice<>C_TENSIONE_FREQUENZA AND
                       i_sys_activedevice<>C_ATTIVAZIONE_V1 AND
                       i_sys_activedevice<>C_DISATTIVAZIONE_V1 AND
                       i_sys_activedevice<>C_IMPOSTA_MANIPOLATORE2D AND
                       i_sys_activedevice<>C_MACCHINA_DX AND
                       i_sys_activedevice<>C_MACCHINA_SX AND
                       i_sys_activedevice<>C_RESET_SIMOTION AND
                       i_sys_activedevice<>C_ON_4RFORM AND
                       i_sys_activedevice<=ULTIMA_OPERAZIONE_COMPLESSA THEN
                      (*dwret:=_restartTaskId(_task.motiontask_CICLI);%%% rewrite with var the action*);
                  END_IF;
              END_IF;
              CURRENT_AXIS:=_FIRST_AXIS#FIRST_AXIS-1;
              CURRENT_STATE:=_FB_MCP483#STATE_MCP483_GEST_JOG_LOOP_STEPS_ELIMINATE_COMMANDS;

          _FB_MCP483#STATE_MCP483_GEST_JOG_LOOP_STEPS_ELIMINATE_COMMANDS:
              IF i_sys_OPMODE=JOGMODE AND i_sys_activedevice<_FIRST_AXIS#FIRST_AXIS THEN
                  CURRENT_STATE:=_FB_MCP483#STATE_MCP483_GEST_JOG_LOOP_AXES_ELIMINATES_TAIL_COMMANDS_LOOP;
              ELSE
                  CURRENT_STATE:=_FB_MCP483#STATE_MCP483_GEST_HOME_ASSI_REALI;
              END_IF;

          _FB_MCP483#STATE_MCP483_GEST_JOG_LOOP_AXES_ELIMINATES_TAIL_COMMANDS_LOOP:

              FOR i:=0 TO _MAXIS#MAXAXIS-1 BY 1 DO
                  IF TestToAttivo(Asse:=i)=TRUE THEN
                    Posax:= AsSynchronousAxisRef(Axes[i].Posax);
                    // Posax:= AsSynchronousAxisRef(UINT#100);
                      IF Posax^.Velocity <>0 THEN //Velocity
                          IF Posax^.StatusWord.%X6 THEN
                          //IF Axes[i].Posax.motionstatedata.motioncommand<>MOTION_DONE THEN
                              CURRENT_STATE:=_FB_MCP483#STATE_MCP483_GEST_JOG_ELIMINATES_CONTROL_LOOP;
                              EXIT;
                          END_IF;
                      END_IF;
                  END_IF;
              END_FOR;
              IF CURRENT_STATE<>_FB_MCP483#STATE_MCP483_GEST_JOG_ELIMINATES_CONTROL_LOOP THEN
                  CURRENT_STATE:=_FB_MCP483#STATE_MCP483_GEST_HOME_ASSI_REALI;
              END_IF;
              (*CURRENT_AXIS:=CURRENT_AXIS+1;
              IF CURRENT_AXIS<_MAXIS#MAXAXIS THEN
                  IF TestToAttivo(Asse:=CURRENT_AXIS)=TRUE THEN
                      IF Axes[CURRENT_AXIS].Posax.motionstatedata.commandvelocity<>0 THEN
                          IF Axes[CURRENT_AXIS].Posax.motionstatedata.motioncommand<>MOTION_DONE THEN
                              CURRENT_STATE:=_FB_MCP483#STATE_MCP483_GEST_JOG_ELIMINATES_CONTROL_LOOP;
                          END_IF;
                      END_IF;
                  END_IF;
              ELSE
                  CURRENT_STATE:=_FB_MCP483#STATE_MCP483_GEST_HOME_ASSI_REALI;
              END_IF;*)

          _FB_MCP483#STATE_MCP483_GEST_JOG_ELIMINATES_CONTROL_LOOP:
              IF EliminaCodaComandi.outputState<>GENERAL_STATE#STATE_END THEN
                  //Arresto assi se rimane attivo un comando ma l^asse è stato disattivato
                  EliminaCodaComandi();
              ELSE
                  EliminaCodaComandi();
                  CURRENT_STATE:=_FB_MCP483#STATE_MCP483_GEST_HOME_ASSI_REALI;
              END_IF;

          _FB_MCP483#STATE_MCP483_GEST_HOME_ASSI_REALI:
              //Gestisce l^HOME solo per assi reali
              IF i_sys_OPMODE=REFMODE THEN
                  IF i_sys_activedevice>=_FIRST_AXIS#FIRST_AXIS THEN
                      IF i_sys_Activedevice<_MAXIS#MAXAXIS+_FIRST_AXIS#FIRST_AXIS THEN
                        If Posax = NULL THEN
                        Posax:= AsSynchronousAxisRef(Axes[i_sys_Activedevice].PosAx);
                        If Posax = NULL THEN;
                        END_IF;
                    END_IF;
                          IF PosAx^.VirtualAxis.Mode = UDINT#0 THEN
                              IF GetEncoderAbsolute(i_sys_Activedevice) THEN
                                  IF mcpi_plus=TRUE THEN
                                      //Serve per poter eseguire l^index dell^asse anche con barriere violate
                                      IF i_sys_accesslevel<=access.index THEN
                                          reset_trace(TRC_LIVELLO_DI_ACCESSO_BASSO);
                                          CURRENT_STATE:=_FB_MCP483#STATE_MCP483_GEST_HOME_HOMING_ABSOLUTE;
                                      ELSE
                                          //Errore livello troppo basso
                                          set_trace(code:=TRC_LIVELLO_DI_ACCESSO_BASSO);
                                      END_IF;
                                  ELSE
                                      CURRENT_STATE:=_FB_MCP483#STATE_MCP483_WATCHDOG_STELIA;
                                  END_IF;
                              ELSE
                                  IF R_PLUS.Q THEN
                                      // lancia task cicli per la presa index di encoder incrementali
                                      CURRENT_STATE:=_FB_MCP483#STATE_MCP483_GEST_HOME_INCREMENTAL_SET_MOVE_AXIS;
                                  ELSE
                                      CURRENT_STATE:=_FB_MCP483#STATE_MCP483_WATCHDOG_STELIA;
                                  END_IF;
                              END_IF;
                          ELSE
                              CURRENT_STATE:=_FB_MCP483#STATE_MCP483_WATCHDOG_STELIA;
                          END_IF;
                      ELSE
                          CURRENT_STATE:=_FB_MCP483#STATE_MCP483_WATCHDOG_STELIA;
                      END_IF;
                  ELSE
                      CURRENT_STATE:=_FB_MCP483#STATE_MCP483_WATCHDOG_STELIA;
                  END_IF;
              ELSE
                  CURRENT_STATE:=_FB_MCP483#STATE_MCP483_WATCHDOG_STELIA;
              END_IF;

          _FB_MCP483#STATE_MCP483_GEST_HOME_HOMING_ABSOLUTE:
              IF Homing_Absolute.outputState<>GENERAL_STATE#STATE_END THEN
                  Homing_Absolute(Asse:=i_sys_activedevice, Position:=pm[i_sys_Activedevice].MA_Refp_Set_Pos);
              ELSE
                  Homing_Absolute();
                  i_sys_chan_request:=1;
                  i_SYS_OPMODE_request:=JOGMODE;
                  CURRENT_STATE:=_FB_MCP483#STATE_MCP483_WATCHDOG_STELIA;
              END_IF;

          _FB_MCP483#STATE_MCP483_GEST_HOME_INCREMENTAL_SET_MOVE_AXIS:
              IF Set_Condizione_Move_Asse.outputState<>GENERAL_STATE#STATE_END THEN
                  SET_Condizione_Move_Asse(Asse:=i_sys_activedevice);
              ELSE
                  SET_Condizione_Move_Asse();
                  IF OK_Condizione_Move_Asse(Asse:=i_sys_activedevice, Direzione:=SN_SP) THEN
                      reset_trace(Code:=TRC_SAFETY_JOG_DEVICES);
                      (*dwret:=_restartTaskId(_task.motiontask_CICLI);*)
                  END_IF;
                  CURRENT_STATE:=_FB_MCP483#STATE_MCP483_WATCHDOG_STELIA;
              END_IF;

          _FB_MCP483#STATE_MCP483_WATCHDOG_STELIA:
              WatchDogStelia();
              CURRENT_STATE:=GENERAL_STATE#STATE_END;

          GENERAL_STATE#STATE_END:
              CURRENT_STATE:=GENERAL_STATE#STATE_INIT;

      END_CASE;
      OutputState:=CURRENT_STATE;
  END_FUNCTION_BLOCK

/**************************************************************************************************
 * WHEN THE TIMER T_NASTRO_FULL EXPIRES, IT CHECKS IF THE FULL BELT INPUT IS STILL ON AND IN THAT *
 *                                CASE IT STOPS THE CONVEYOR BELT                                 *
 **************************************************************************************************/
(*{
#ifndef ORBITALE
}*)
	FUNCTION ArrestoNastroPieno

        VAR_EXTERNAL
            TimerSistema                    :ARRAY[0..MAX_TIMER_SISTEMA-1] OF Timer;
            OAddress                        : ARRAY [0..MAXDIGITALOUTPUT] OF Digital_Output;
        	Clk_NastroPieno					:BOOL;
	        R_NastroPieno							:R_TRIG;	//Fronte salita nastro trasportatore pieno
            TimeNastFull				    :INT;
        END_VAR

        VAR_EXTERNAL CONSTANT
            MAX_TIMER_SISTEMA 	        :USINT;
            MAXDIGITALOUTPUT            :INT;
            T_NAST_FULL 				:INT;
            OUT_NAST_TRANSPORTER        :INT;
            INP_NAST_TRANSPORTER_FULL	:INT;
        END_VAR

		Clk_NastroPieno:=TimerSistema[T_NAST_FULL].Executed;
		R_NastroPieno(clk:=Clk_NastroPieno);
		IF R_NastroPieno.q=TRUE AND ReadDigitalInput(NumInput:=INP_NAST_TRANSPORTER_FULL)=TRUE THEN
			ComandoNastroTrasportatore(Stato:=FALSE);
		END_IF;
		IF ReadDigitalInput(NumInput:=INP_NAST_TRANSPORTER_FULL)=TRUE AND
			 TimerSistema[T_NAST_FULL].Status=0 AND
			 OAddress[OUT_NAST_TRANSPORTER].Stato=TRUE THEN
			//Partenza timer se è attivo l^ingresso di nastro pieno e l^uscita di comando del nastro
			TimerSistema[T_NAST_FULL].Value:=TimeNastFull;
			TimerSistema[T_NAST_FULL].Status:=SINT#1;
		END_IF;
	END_FUNCTION
(*{
#endif	//Fine NO ORBITALE
}*)

/******************************************************************************************
 * PERFORMS SELECTION MANAGEMENT VIA PNPN OR DPDP OF THE PRODUCTION TABLE TO BE ACTIVATED *
 ******************************************************************************************/

FUNCTION GestioneTabelleProduzione

    VAR_EXTERNAL
        i_sys_OPMODE                    : INT;	// MODO OPERATIVO
                                                // 0 = JOG
                                                // 1 = REFERENCE
                                                // 2 = MDA
                                                // 3 = AUTO
        DatiSelExtProd					:SelExtProd;
        F_InpCodiceTabellaOK	        :F_TRIG; //fronte discesa InpCodiceTabellaOK
    END_VAR

    VAR_EXTERNAL CONSTANT
        JOGMODE                               :INT;
    END_VAR
	VAR
		AppoOutCodiceTabellaOK    :BOOL:=FALSE;
		AppoCodiceErroreTabExt    :INT:=0;
		i                                                :INT;
	END_VAR
	IF i_sys_OPMODE=JOGMODE AND DatiSelExtProd.AbilSelExtTabella=TRUE THEN
		//Lettura dal bus di campo delle informazioni provenienti dal supervisore
		LetturaDatiTabellaProduzione(CodiceTabella:=DatiSelExtProd.CodiceTabellaDaCaricare,
																 AbilPezSegTabExt:=DatiSelExtProd.AbilPezSegTabExt,
																 InpCodiceTabellaOK:=DatiSelExtProd.InpCodiceTabellaOK);
		//Abilitazione sorveglianza sul cambio di stato del segnale di strobe di convalida
		F_InpCodiceTabellaOK(clk:=DatiSelExtProd.InpCodiceTabellaOK);
		IF F_InpCodiceTabellaOK.q=TRUE THEN
			//Il fronte di discesa della variabile "InpCodiceTabellaOK" indica che la codifica della tabella di produzione non è più coerente.
			//Quindi si resetta la variabile "OutCodiceTabellaOK" che indica al supervissore lo stato della tabella di produzione.
			DatiSelExtProd.OutCodiceTabellaOK:=FALSE;
			//Si resetta (-1) anche il codice di un eventuale errore di attivazione della tabella di produzione
			DatiSelExtProd.CodiceErroreTabExt:=-1;
		END_IF;
		IF DatiSelExtProd.CodiceErroreTabExt=0 THEN
			DatiSelExtProd.OutCodiceTabellaOK:=TRUE;
		ELSE
			IF DatiSelExtProd.CodiceErroreTabExt>0 THEN
				//In caso di errore viene resetta la variabile che indica che la tabella di produzione richiesta è stata trasferita al Simotion
				DatiSelExtProd.OutCodiceTabellaOK:=FALSE;
				//Invalida i dati dei pezzi in quanto dovrà essere inviata la produzione
				InvalidaProgrammi();
			END_IF;
		END_IF;
		IF DatiSelExtProd.InpCodiceTabellaOK=FALSE THEN
			DatiSelExtProd.OutCodiceTabellaOK:=FALSE;
		END_IF;
		ScritturaDatiTabellaProduzione(CodiceErroreTabExt:=DatiSelExtProd.CodiceErroreTabExt, OutCodiceTabellaOK:=DatiSelExtProd.OutCodiceTabellaOK);
	ELSE
		AppoOutCodiceTabellaOK:=FALSE;
		AppoCodiceErroreTabExt:=0;
		ScritturaDatiTabellaProduzione(CodiceErroreTabExt:=AppoCodiceErroreTabExt, OutCodiceTabellaOK:=AppoOutCodiceTabellaOK);
	END_IF;
END_FUNCTION

/**********************************************************************************************************************
 *                  VIA DPDP OR PNPN READS THE FOLLOWING INFORMATION WHICH IS SET BY THE SUPERVISOR:                  *
 *                  -BYTE X05 (LOW) AND X06(HIGH) => NUMBER OF THE PRODUCTION TABLE TO BE ACTIVATED                   *
 *               -BYTE X04 BIT 0 => STROBE TO VALIDATE THE CODE OF THE PRODUCTION TABLE TO BE ACTIVATED               *
 * -BYTE X04 BIT 1 => TRUE IN THE ACTIVE TABLE ENABLES THE FOLLOWING WORKPIECE MODE, FALSE ENABLES EXTERNAL SELECTION *
 **********************************************************************************************************************/

FUNCTION LetturaDatiTabellaProduzione

    VAR_EXTERNAL
        i_sys_DpCoupler                 :BOOL;
        V_pncoupler_i                   : pncoupler_i;
        V_dbcoupler_i                   : dbcoupler_i;
        i_sys_PnCoupler                 :BOOL;
    END_VAR

	VAR_IN_OUT
		CodiceTabella			:DINT;	//Numero della tabella di produzione che deve essere attivata
		AbilPezSegTabExt	    :BOOL;	//TRUE abilita il pezzo seguente, FALSE abilita la selezione esterna
		InpCodiceTabellaOK      :BOOL;	//Strobe di convalida dei dati di input
	END_VAR

    VAR
		AppoByteBasso	:WORD;
		AppoByteAlto	:WORD;
        tmpword:word;
	END_VAR
	// {
	// #ifndef EMULAZIONE
	// }
		AppoByteBasso:=WORD#0;
		AppoByteAlto:=WORD#0;
		IF i_sys_DpCoupler=TRUE THEN
			AppoByteBasso:=V_dbcoupler_i.address_db_i[5];
			AppoByteAlto:=V_dbcoupler_i.address_db_i[6];
			InpCodiceTabellaOK:=getbit(V_dbcoupler_i.address_db_i[4], USINT#0);
			AbilPezSegTabExt:=getbit(V_dbcoupler_i.address_db_i[4], USINT#1);
		ELSE
			// {
			// #ifdef PROFINET
			// }
				IF i_sys_PnCoupler=TRUE THEN
					AppoByteBasso:=V_pncoupler_i.address_pn_i[5];
					AppoByteAlto:=V_pncoupler_i.address_pn_i[6];
					InpCodiceTabellaOK:=getbit(V_pncoupler_i.address_pn_i[4], USINT#0);
					AbilPezSegTabExt:=getbit(V_pncoupler_i.address_pn_i[4], USINT#1);
				END_IF;
			// {
			// #endif	//Fine PROFINET
			// }
			;
		END_IF;

		CodiceTabella:=TO_DINT(SHL(AppoByteAlto,uint#8) or AppoByteBasso);

	// {
	// #endif	//Fine NO EMULAZIONE
	// }
	;
END_FUNCTION

/*****************************************************************************************************
 *            WRITES INFORMATION TO DPDP OR PNPN WHICH IS TRANSFERRED TO THE SUPERVISOR:             *
 * -BYTE X42 BIT 3 => TRUE THE PRODUCTION TABLE CANNOT BE ACTIVATED DUE TO AN ERROR INDICATED BY VGP *
 *      -BYTE X42 BIT 5 => TRUE THE PRODUCTION TABLE HAS BEEN ACTIVATED AND NO ERROR IS PRESENT      *
 *****************************************************************************************************/
(* *)
FUNCTION ScritturaDatiTabellaProduzione

    VAR_EXTERNAL
        i_sys_DpCoupler                 :BOOL;
        i_sys_PnCoupler                 :BOOL;
        V_pncoupler_o                   : pncoupler_o;
        V_dbcoupler_o                   : dbcoupler_o;

    END_VAR

	VAR_IN_OUT
		CodiceErroreTabExt	:INT;		//True errore nell^attivazione della tabella di produzione, False nessun errore
		OutCodiceTabellaOK	:BOOL;	//True la tabella di produzione è stata attivata
	END_VAR

    VAR_TEMP
        Local_dbcoupler_o42                   : BYTE;
        Local_pncoupler_o42                   : BYTE;
    END_VAR
	IF i_sys_DpCoupler=TRUE THEN
        Local_dbcoupler_o42:=V_dbcoupler_o.address_db_o[42];
		V_dbcoupler_o.address_db_o[42]:=setbit(Local_dbcoupler_o42, USINT#3, TO_BOOL(MAX(0,CodiceErroreTabExt)));
	ELSE
		// {
		// #ifdef PROFINET
		// }
			IF i_sys_PnCoupler=TRUE THEN
                Local_pncoupler_o42:=V_pncoupler_o.address_pn_o[42];
				V_pncoupler_o.address_pn_o[42]:=setbit(Local_pncoupler_o42, USINT#3, TO_BOOL(MAX(0,CodiceErroreTabExt)));
				V_pncoupler_o.address_pn_o[42]:=setbit(Local_pncoupler_o42, USINT#5, OutCodiceTabellaOK);
			END_IF;
		// {
		// #endif    //Fine PROFINET
		// }
		;
	END_IF;
END_FUNCTION

// {
// #ifdef DH4010
// }
	FUNCTION TestCicloSpedizioneEseguito:BOOL

    VAR_EXTERNAL
        pm                              : ARRAY[_FIRST_AXIS#FIRST_AXIS.._FIRST_AXIS#FIRST_AXIS+_CONST_VAR_DEF._MAXIS#MAXAXIS-1] OF AxisParameters;
        Axes                            :ARRAY[_FIRST_AXIS#FIRST_AXIS.._FIRST_AXIS#FIRST_AXIS+_CONST_VAR_DEF._MAXIS#MAXAXIS-1] OF ax;/// ax as structure is defined in _TYPE
        i_sys_CicloSpedizioneEseguito   :BOOL;     //True se è stato eseguito il ciclo di spedizione
    END_VAR

    VAR_EXTERNAL CONSTANT

        X1:INT;
        X2:INT;
    END_VAR

    VAR
        PosAx : REF_TO TO_SynchronousAxis;
    END_VAR

        PosAx:= AsSynchronousAxisRef(Axes[X2].PosAx);
		// IF (ABS(pm[X2].MA_Spedizione_BLM-PosAx^.actualPosition)<pm[X2].MA_Tolerance AND   //takeBack
		// 		pm[X2].MA_Spedizione_BLM<pm[X2].Ma_Pos_Limit_Minus AND pm[X2].MA_Spedizione_BLM>pm[X2].Ma_Pos_Limit_Plus) OR
		// 	 i_sys_CicloSpedizioneEseguito=TRUE THEN
		// 	TestCicloSpedizioneEseguito:=TRUE;
		// ELSE
		// 	TestCicloSpedizioneEseguito:=FALSE;
		// END_IF;
        // PosAx:= AsSynchronousAxisRef(Axes[X1].PosAx);
		// IF (ABS(pm[X1].MA_Spedizione_BLM-PosAx^.actualPosition)<pm[X1].MA_Tolerance AND
		// 		pm[X1].MA_Spedizione_BLM<pm[X1].Ma_Pos_Limit_Minus AND pm[X1].MA_Spedizione_BLM>pm[X1].Ma_Pos_Limit_Plus) OR
		// 		i_sys_CicloSpedizioneEseguito=TRUE THEN
		// 	TestCicloSpedizioneEseguito:=TRUE;
		// ELSE
		// 	TestCicloSpedizioneEseguito:=FALSE;
		// END_IF;
	END_FUNCTION

/******************************************************************************************************
 * RETURNS TRUE IF IT IS INTENDED THAT THE MOVEMENT IN JOG OF THE DEVICE PASSED AS A PARAMETER CAN BE *
 *                              ASSOCIATED WITH A POSITIONING OF AN AXIS                              *
 ******************************************************************************************************/
FUNCTION TestDispConAsse:BOOL

    VAR_EXTERNAL CONSTANT
        Z1:INT;
        PALETTA                               :INT;
    END_VAR

	VAR_INPUT
		Disp    :INT;
		Asse    :INT;
	END_VAR
	TestDispConAsse:=FALSE;
	// // { %%%%
	// // #ifdef ORBITALE
	// // }
	// // 	{
	// // 	#ifdef DH4010
	// // 	}
	// 		IF Disp=SCOMP_MANIPOLATORE_3D AND Asse=Z1 THEN
	// 			//Il dispositivo SCOMP_MANIPOLATORE_3D per potersi muovere deve prima posizionare a 65° l^asse Z1
	// 			TestDispConAsse:=TRUE;
	// 		END_IF;
	// // 	{
	// // 	#endif  //Fine DH4010
	// // 	}
	// // {
	// // #else    //Fine ORBITALE
	// // }
		IF Disp=PALETTA AND Asse=Z1 THEN
			//Il dispositivo PALETTA per potersi muovere deve prima posizionare a 0° l^asse Z1
			TestDispConAsse:=TRUE;
		END_IF;
	// {
	// #endif  //Fine NO ORBITALE
	// }
END_FUNCTION

    FUNCTION WatchdogStelia

        VAR_EXTERNAL
            OAddress                        : ARRAY [0..MAXDIGITALOUTPUT] OF Digital_Output;
        END_VAR

        VAR_EXTERNAL CONSTANT
            MAXDIGITALOUTPUT                    :INT;
            OUT_01_STOP_POINT                             :INT;
            OUT_02_STOP_POINT                             :INT;
            OUT_03_STOP_POINT                             :INT;
            OUT_04_STOP_POINT                             :INT;

            INP_01_STOP_POINT                           :INT;
            INP_02_STOP_POINT                           :INT;
            INP_03_STOP_POINT                           :INT;
        END_VAR

        VAR
          iret  :INT;
        END_VAR
        ;
        // IF i_sys_CM_1243_5=TRUE THEN
        // //   {
        // //   #ifdef ELECTM
        // //   }
        // //     {
        // //     #ifndef PROFINET
        // //     }
        //       o_defects_acknoledge:=mcpi_reset;
        //       o_transmitters_1_2_used:=OAddress[OUT_01_STOP_POINT].stato;
        //       o_transmitters_3_4_used:=OAddress[OUT_02_STOP_POINT].stato;
        //       o_transmitters_5_6_used:=OAddress[OUT_03_STOP_POINT].stato;
        //               (* Tolte in base al documento di Stelia inviato con email di Luca Proserpio di martedì 03/10/2017 16:50
        //                   o_transmitters_7_8_used:=OAddress[OUT_04_STOP_POINT].stato;
        //                   o_override:=LREAL_VALUE_TO_BYTE(i_sys_hwovr);
        //                   o_machine_state:=LREAL_VALUE_TO_WORD(Protube.MachineState.MachineState);
        //               *)
        //       IAddress[INP_01_STOP_POINT].enable_forzatura:=TRUE;
        //       IAddress[INP_01_STOP_POINT].stato_forzatura:=i_temperature_ok;
        //       IF i_running_mode<1 OR i_running_mode>2 THEN
        //         IF i_sys_error<>ERR_HEATING_MODE THEN
        //           iret:=Push_error(code:=ERR_HEATING_MODE, Arresto:=FALSE);
        //         END_IF;
        //       END_IF;
        //       IF i_general_defect=TRUE THEN
        //         IF i_sys_error<>ERR_HEATING_ERROR THEN
        //           iret:=Push_error(code:=ERR_HEATING_ERROR, Arresto:=FALSE);
        //         END_IF;
        //       END_IF;
        //       IF EnableWatchdog=TRUE THEN
        //         o_watchdog:=i_watchdog;
        //         IF Old_I_WatchDog=i_watchdog THEN
        //           //Valore non cambiato si verifica che il timer non sia arrivato
        //           //a zero, altrimenti errore
        //           IF TimerSistema[T_WATCHDOG].valore<1 THEN
        //             IF i_sys_error<>ERR_WATCHDOG THEN
        //               iret:=Push_error(code:=ERR_WATCHDOG, Arresto:=FALSE);
        //             END_IF;
        //           END_IF;
        //         ELSE
        //           //Input cambiato si fa ripartire il timer (1 sec)
        //           Old_I_WatchDog:=o_watchdog;
        //           TimerSistema[T_WATCHDOG].valore:=1000;
        //           TimerSistema[T_WATCHDOG].stato:=1;
        //         END_IF;
        //       ELSE
        //         IF i_watchdog=TRUE THEN
        //           //Il watchdog parte alla prima attivazione di i_watchdog
        //           EnableWatchdog:=TRUE;
        //         END_IF;
        //       END_IF;
        //               //Copia variabili su area di scambio
        //               Heating.input.working_status:=i_working_status;
        //               Heating.input.running_mode:=i_running_mode;
        //               Heating.input.temperature_measurement:=i_temperature_measurement;
        //               Heating.input.pyrometer_position_measurement:=i_pyrometer_position_measurement;
        //               Heating.input.general_defect:=i_general_defect;
        //               Heating.input.watchdog:=i_watchdog;
        //               Heating.input.temperature_ok:=i_temperature_ok;
        //               Heating.output.temperature_setpoint:=o_temperature_setpoint;
        //               Heating.output.tube_diameter:=o_tube_diameter;
        //               Heating.output.first_heat:=o_first_heat;
        //               Heating.output.last_heat:=o_last_heat;
        //               Heating.output.defects_acknoledge:=o_defects_acknoledge;
        //               Heating.output.watchdog:=o_watchdog;
        //               Heating.output.transmitters_1_2_used:=o_transmitters_1_2_used;
        //               Heating.output.transmitters_3_4_used:=o_transmitters_3_4_used;
        //               Heating.output.transmitters_5_6_used:=o_transmitters_5_6_used;
        //               Heating.output.transmitters_7_8_used:=OAddress[OUT_04_STOP_POINT].stato;
        //               Heating.output._override:=LREAL_VALUE_TO_BYTE(i_sys_hwovr);
        //               Heating.output.machine_state:=LREAL_VALUE_TO_WORD(Protube.MachineState.MachineState);
        // //     {
        // //     #endif  //Fine NO PROFINET
        // //     }
        // //   {
        // //   #endif  //Fine ELECTM
        // //   }
        // //   ;
        // END_IF;

      END_FUNCTION

  END_NAMESPACE
